FUNCTION_BLOCK FB_CTD_UDINT (* Down counter *)
  PACKAGE iec61131::counters;
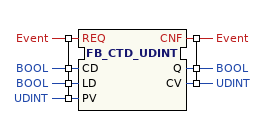
  EVENT_INPUT
    REQ WITH CD, PV, LD; (* Normal Execution Request *)
  END_EVENT
  EVENT_OUTPUT
    CNF WITH Q, CV; (* Execution Confirmation *)
  END_EVENT
  VAR_INPUT
    CD : BOOL; (* Count down *)
    LD : BOOL; (* Load *)
    PV : UDINT; (* Preset value *)
  END_VAR
  VAR_OUTPUT
    Q : BOOL; (* Output *)
    CV : UDINT; (* Count value *)
  END_VAR
  ALGORITHM REQ IN ST:
IF LD THEN
  CV := PV;
ELSIF CD AND CV> 0 THEN
  CV := CV - 1;
END_IF;
Q := CV <= 0;
  END_ALGORITHM
END_FUNCTION_BLOCK
